(* PLC project Tc3_EventLogger.HRESULTAdsErr_TO_TcEventEntry Demo, tc3-libraries-kb TwinCAT 3.1 *)
(* stored: creationDateTime 2026-05-11T01:00:00, modificationDateTime 2026-05-11T01:00:00 *)

PROGRAM P_Demo_HRESULTAdsErr_TO_TcEventEntry
  VAR
    hr : E_HRESULTAdsErr := E_HRESULTAdsErr.HRESULTADSERR_DEVICE_INVALIDPARM;  (* 在线写入要转换的 HRESULT 错误码 *)
    stEventEntry : TcEventEntry;  (* 转换输出 *)
    bOk : BOOL;  (* 成功标志 *)
  END_VAR

// =============================================================================
// 场景：HRESULT ADS 错误码 → TcEventEntry 转换
// 价值：HRESULT 形式 ADS 错的归一化
// 验证：登录后给输入赋已知合法值；调用本 FC 后 bOk 应为 TRUE 且输出已填
// 验证步骤：
//   1. 右键 PLC 项目 → Import PLCopenXML → 选本文件
//   2. 引用 Tc3_EventLogger（System → References → Add library）
//   3. 编译 → 登录 → 运行；按 verify 注释里给出的在线写值操作
// =============================================================================

bOk := HRESULTAdsErr_TO_TcEventEntry(
    hr := hr,
    stEventEntry := stEventEntry);
END_PROGRAM
